// TIA Portal V16 export
// export: Created 2022-02-28T20:47:28.8923176Z, ExportSetting WithDefaults, DisplayName Totally Integrated Automation Portal, DisplayVersion V16, DisplayName TIA Portal Version Control Interface, DisplayVersion V16, DisplayName TIA Portal Openness, DisplayVersion V16, DisplayName STEP 7 Professional, DisplayVersion V16, DisplayName STEP 7 Safety, DisplayVersion V16, DisplayName WinCC Advanced, DisplayVersion V16
VAR_GLOBAL   // PLC tag table "03_Camara_2"
   "DataMan2-TriggerEnable" AT %Q73.0 : Bool;
   "DataMan2-Trigger" AT %Q73.1 : Bool;
   "DataMan2-TriggerReady" AT %I79.0 : Bool;
   "DataMan2-TriggerAck" AT %I79.1 : Bool;
   "DataMan2-Acquiring" AT %I79.2 : Bool;
   "DataMan2-MissedAcq" AT %I79.3 : Bool;
   "DataMan2-TriggerID" AT %IW80 : Word;
   "DataMan2-BufferResultsEnable" AT %Q74.0 : Bool;
   "DataMan2-ResultsAck" AT %Q74.1 : Bool;
   "DataMan2-Decoding" AT %I82.0 : Bool;
   "DataMan2-Decode Complete" AT %I82.1 : Bool;
   "DataMan2-Results Buffer Overrun" AT %I82.2 : Bool;
   "DataMan2-Results Available" AT %I82.3 : Bool;
   "DataMan2-General Fault" AT %I82.7 : Bool;
   "DataMan2-Train Code" AT %Q75.0 : Bool;
   "DataMan2-Train Match String" AT %Q75.1 : Bool;
   "DataMan2-Train Focus" AT %Q75.2 : Bool;
   "DataMan2-Train Brightness" AT %Q75.3 : Bool;
   "DataMan2-Untrain" AT %Q75.4 : Bool;
   "DataMan2-Execute DMCC" AT %Q75.6 : Bool;
   "DataMan2-Set Match String" AT %Q75.7 : Bool;
   "DataMan2-Train Code Ack" AT %I83.0 : Bool;
   "DataMan2-Train Match String Ack" AT %I83.1 : Bool;
   "DataMan2-Train Focus Ack" AT %I83.2 : Bool;
   "DataMan2-Train Brightness Ack" AT %I83.3 : Bool;
   "DataMan2-Untrain Ack" AT %I83.4 : Bool;
   "DataMan2-Execute DMCC Ack" AT %I83.6 : Bool;
   "DataMan2-Set Match String Ack" AT %I83.7 : Bool;
   "DataMan2-UserData Option" AT %QW76 : Word;
   "DataMan2-UserData Length" AT %QW78 : Word;
   "DataMan2-UserData[0]" AT %QB80 : Byte;
   "DataMan2-UserData[1]" AT %QB81 : Byte;
   "DataMan2-UserData[2]" AT %QB82 : Byte;
   "DataMan2-UserData[3]" AT %QB83 : Byte;
   "DataMan2-UserData[4]" AT %QB84 : Byte;
   "DataMan2-UserData[5]" AT %QB85 : Byte;
   "DataMan2-UserData[6]" AT %QB86 : Byte;
   "DataMan2-UserData[7]" AT %QB87 : Byte;
   "DataMan2-UserData[8]" AT %QB88 : Byte;
   "DataMan2-UserData[9]" AT %QB89 : Byte;
   "DataMan2-UserData[10]" AT %QB90 : Byte;
   "DataMan2-UserData[11]" AT %QB91 : Byte;
   "DataMan2-UserData[12]" AT %QB92 : Byte;
   "DataMan2-UserData[13]" AT %QB93 : Byte;
   "DataMan2-UserData[14]" AT %QB94 : Byte;
   "DataMan2-UserData[15]" AT %QB95 : Byte;
   "DataMan2-ResultID" AT %IW84 : Word;
   "DataMan2-Result Code" AT %IW86 : Word;
   "DataMan2-Result Extended" AT %IW88 : Word;
   "DataMan2-Result Length" AT %IW90 : Word;
   "DataMan2-InspectionResults[0]" AT %IB92 : Byte;
   "DataMan2-InspectionResults[1]" AT %IB93 : Byte;
   "DataMan2-InspectionResults[2]" AT %IB94 : Byte;
   "DataMan2-InspectionResults[3]" AT %IB95 : Byte;
   "DataMan2-InspectionResults[4]" AT %IB96 : Byte;
   "DataMan2-InspectionResults[5]" AT %IB97 : Byte;
   "DataMan2-InspectionResults[6]" AT %IB98 : Byte;
   "DataMan2-InspectionResults[7]" AT %IB99 : Byte;
   "DataMan2-InspectionResults[8]" AT %IB100 : Byte;
   "DataMan2-InspectionResults[9]" AT %IB101 : Byte;
   "DataMan2-InspectionResults[10]" AT %IB102 : Byte;
   "DataMan2-InspectionResults[11]" AT %IB103 : Byte;
   "DataMan2-InspectionResults[12]" AT %IB104 : Byte;
   "DataMan2-InspectionResults[13]" AT %IB105 : Byte;
   "DataMan2-InspectionResults[14]" AT %IB106 : Byte;
   "DataMan2-InspectionResults[15]" AT %IB107 : Byte;
END_VAR
